FUNCTION_BLOCK FB_HeaterProtection
VAR_INPUT
	Excute:BOOL;
END_VAR
VAR_OUTPUT
	Done:BOOL;
	Busy:BOOL;
END_VAR
VAR
	Timer:TON;
	Step:INT;
END_VAR


IF Excute THEN
	Step:= 10;
	Done:=FALSE;
	Excute:=FALSE;
	Busy:=TRUE;
	
	
END_IF

CASE Step OF

	0://wait
	
	10:
		Timer.PT := DINT_TO_TIME( Persist.PersistentStruct.TimerHotWeldingOn);
		Timer.IN:=TRUE;
		gMachineCtrl.IO.Out.HeaterOn:=TRUE;
		IF Timer.Q THEN
			gMachineCtrl.IO.Out.HeaterOn:=FALSE;
			Step:=20;
		END_IF
	
	20:
		Done:=TRUE;
		Timer.IN:=FALSE;
		Busy:=FALSE;
	
END_CASE

Timer();

END_FUNCTION_BLOCK

(* stored: Version 1.1.0.1, ProductVersion 3.1.4024.3
   POU FB_HeaterProtection: Id {fd0095b0-37d0-4488-85cb-9454a8330829}, SpecialFunc None *)
